# EPICS substitutions: epics/db/EL2032.substitutions
file "./db/ecSlave.template"
{
  pattern {}
          {}
}

# No custom data yet
#file "./db/EL2032.template"
#{
#  pattern {}
#          {}
#}
